// TwinCAT 3 PLC project MainPLC
// ProgramVersion: 3.1.4024.0
// libraries:
//   Tc2_Standard, * (Beckhoff Automation GmbH)
//   Tc2_System, * (Beckhoff Automation GmbH)
//   Tc3_Module, * (Beckhoff Automation GmbH)
// project tree:
//   / PlcTask.TcTTO
//   POUs/ FU_Conveyor.TcPOU, MAIN.TcPOU

CONFIGURATION MainPLC
    RESOURCE PLC ON TwinCAT3
        TASK PlcTask(INTERVAL := T#10ms, PRIORITY := 20);
        PROGRAM MAIN WITH PlcTask : MAIN;
    END_RESOURCE
END_CONFIGURATION

// ---- POUs/MAIN.TcPOU
PROGRAM MAIN
VAR
END_VAR

END_PROGRAM

// ---- POUs/FU_Conveyor.TcPOU
FUNCTION_BLOCK FU_Conveyor
VAR_INPUT
END_VAR
VAR_OUTPUT
END_VAR
VAR
	Sensor : BOOL;
	PrevSensor : BOOL;
	Motor : BOOL;
	Timer1 : TON;
END_VAR

IF Sensor AND NOT PrevSensor THEN
	Motor := TRUE;
END_IF

Timer1(IN := Motor, PT := T#3S);

IF Timer1.Q THEN
	Motor := FALSE;
END_IF

PrevSensor := Sensor;

END_FUNCTION_BLOCK
